// TIA Portal V19 export
DATA_BLOCK "HEADER_DATA"   // DB170
{ S7_Optimized_Access := 'TRUE' }
// stored: MemoryReserve 100
BEGIN
END_DATA_BLOCK
